// TIA Portal V17 export
// export: Created 2024-09-02T12:50:04.2483482Z, ExportSetting WithDefaults, DisplayName Totally Integrated Automation Portal, DisplayVersion V17, DisplayName TIA Portal Openness, DisplayVersion V17, DisplayName TIA Portal Version Control Interface, DisplayVersion V17, DisplayName STEP 7 Professional, DisplayVersion V17, DisplayName STEP 7 Safety, DisplayVersion V17, DisplayName WinCC Professional, DisplayVersion V17
FUNCTION "SysFC_RF300_Comunication" : Void   // FC801, LAD
TITLE = RF300 Commands / RF300 Befehle
{ S7_Optimized_Access := 'TRUE' }
AUTHOR : STEAM
FAMILY : MOBY
NAME : MOBY
VERSION : 0.1
// stored: AutoNumber true, IsIECCheckEnabled false, SetENOAutomatically false, UDAEnableTagReadback false
   VAR_INPUT
      SequenceNr : Int;   // Sequenznummer des Funktionsaufrufes (muss Eindeutig pro SLG sein) / Sequence number of function call (must be unique for each SLG)
      FunctionNr : Int;   // Funktionsanwahl 1 - lesen, 2- schreiben usw. / Function selection 1 - read, 2- write etc.
      Start : Bool;   // Funktionsanwahl "Lesen" / function selection "Read"
      Reset : Bool;
      ADR_MDS : Int;   // Adresse Datenträger (MDS) / Data carrier address (MDS)
      ByteLength : Int;   // Anzahl der Bytes / Number of bytes
   END_VAR
   VAR_OUTPUT
      FunktionOk : Bool;
   END_VAR
   VAR_IN_OUT
      MDS_Data : Variant;
      Command : "TypeMobyBefehle";
      Finish : Bool;   // Auftrag Fertig "Lesen / Order Finished "Read"
   END_VAR
   VAR_TEMP
      t_VKE0 : Bool;
      t_VKE1 : Bool;
      t_RetVal : Word;
      t_OrderLineReady : Bool;
      t_MainOrderReady : Bool;
      t_FaultBuffer : Bool;
      t_HugeBuffer : UDInt;
      t_TempDInt : DInt;
      t_Command_INIT : "TypeMobySequenz";
   END_VAR
   VAR_TEMP   // added for the SCL form of the ladder/FBD networks
      _w1 : Bool;
      _w2 : Bool;
      _w3 : Bool;
   END_VAR
BEGIN

REGION Network 1: INIT
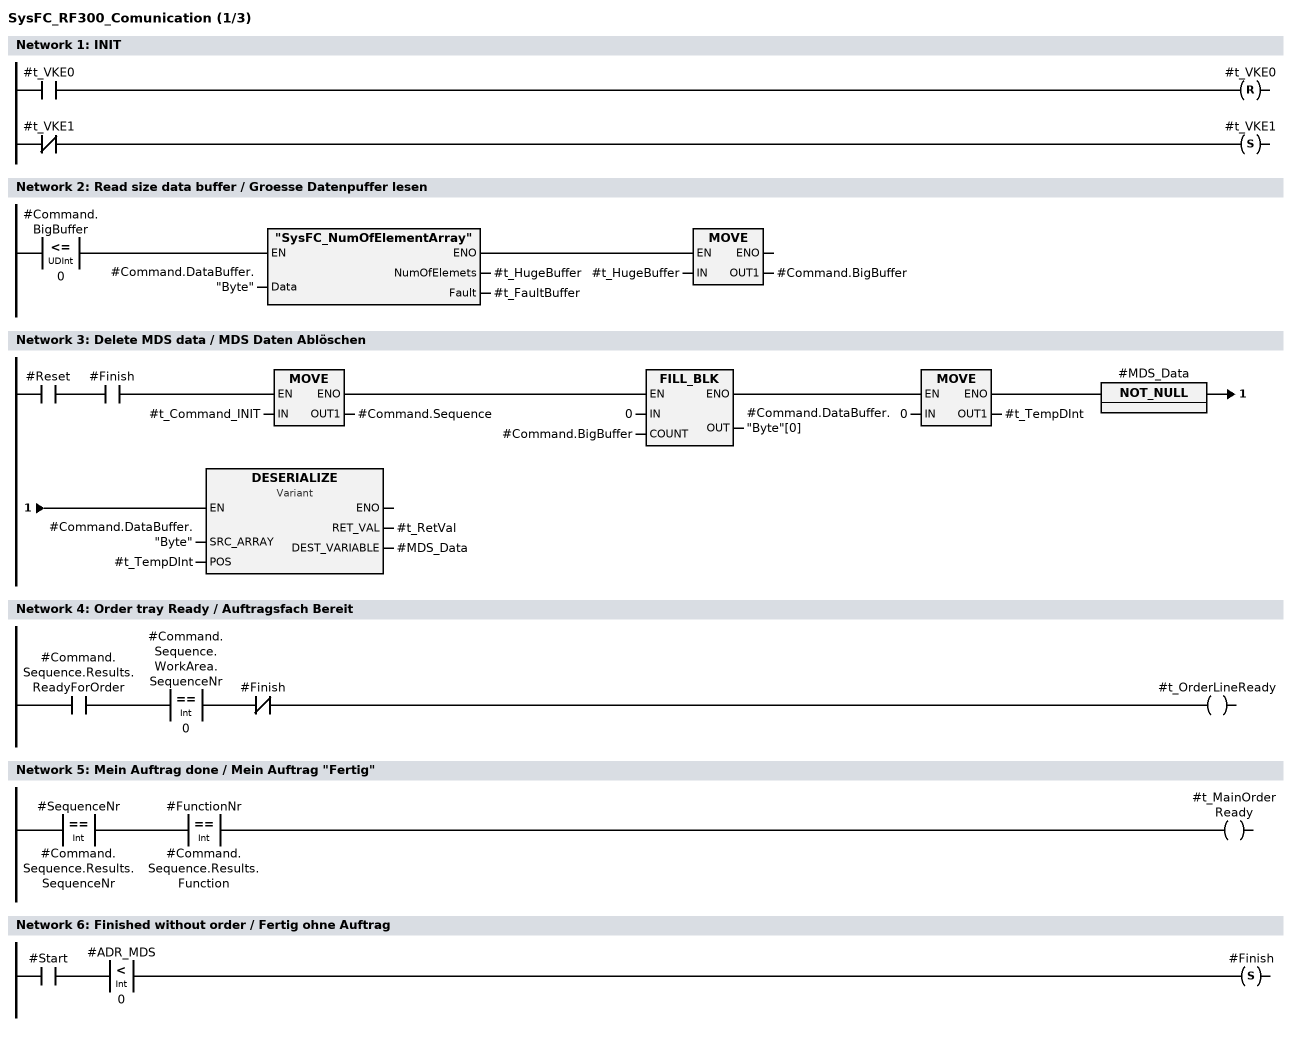
   RUNG wire#powerrail
      Contact( #t_VKE0 )
      R_Coil( #t_VKE0 )
   END_RUNG
   RUNG wire#powerrail
      I_Contact( #t_VKE1 )
      S_Coil( #t_VKE1 )
   END_RUNG
   // the same network as SCL:
   IF #t_VKE0 THEN #t_VKE0 := FALSE; END_IF;
   IF NOT #t_VKE1 THEN #t_VKE1 := TRUE; END_IF;
END_REGION

REGION Network 2: Read size data buffer / Groesse Datenpuffer lesen
   RUNG wire#powerrail
      { S7_Templates := "SrcType := UDInt" } LE_Contact(in1 := #Command.BigBuffer, in2 := 0)
      "SysFC_NumOfElementArray"(Data := #Command.DataBuffer."Byte", NumOfElemets => #t_HugeBuffer, Fault => #t_FaultBuffer)
      Move(in := #t_HugeBuffer, out1 => #Command.BigBuffer)
   END_RUNG
   // the same network as SCL:
   "SysFC_NumOfElementArray"(EN := #Command.BigBuffer <= 0,
                           Data := #Command.DataBuffer."Byte",
                           NumOfElemets => #t_HugeBuffer,
                           Fault => #t_FaultBuffer,
                           ENO => #_w1);
   IF #_w1 THEN #Command.BigBuffer := #t_HugeBuffer; END_IF;
END_REGION

REGION Network 3: Delete MDS data / MDS Daten Ablöschen
   // no SCL statement known for NOT_NULL: written as a call
   #_w1 := #Reset AND #Finish;
   IF #_w1 THEN
       #Command.Sequence := #t_Command_INIT;
       FILL_BLK(IN := 0, COUNT := #Command.BigBuffer, OUT => #Command.DataBuffer."Byte"[0]);
       #t_TempDInt := 0;
   END_IF;
   IF #_w1 AND NOT_NULL(#MDS_Data) THEN
       #t_RetVal := Deserialize(SRC_ARRAY := #Command.DataBuffer."Byte",
                               POS := #t_TempDInt,
                               DEST_VARIABLE => #MDS_Data);
   END_IF;
END_REGION

REGION Network 4: Order tray Ready / Auftragsfach Bereit
   RUNG wire#powerrail
      Contact( #Command.Sequence.Results.ReadyForOrder )
      { S7_Templates := "SrcType := Int" } EQ_Contact(in1 := #Command.Sequence.WorkArea.SequenceNr, in2 := 0)
      I_Contact( #Finish )
      Coil( #t_OrderLineReady )
   END_RUNG
   // the same network as SCL:
   #t_OrderLineReady := #Command.Sequence.Results.ReadyForOrder AND (#Command.Sequence.WorkArea.SequenceNr = 0) AND NOT #Finish;
END_REGION

REGION Network 5: Mein Auftrag done / Mein Auftrag "Fertig"
   RUNG wire#powerrail
      { S7_Templates := "SrcType := Int" } EQ_Contact(in1 := #SequenceNr, in2 := #Command.Sequence.Results.SequenceNr)
      { S7_Templates := "SrcType := Int" } EQ_Contact(in1 := #FunctionNr, in2 := #Command.Sequence.Results.Function)
      Coil( #t_MainOrderReady )
   END_RUNG
   // the same network as SCL:
   #t_MainOrderReady := (#SequenceNr = #Command.Sequence.Results.SequenceNr) AND (#FunctionNr = #Command.Sequence.Results.Function);
END_REGION

REGION Network 6: Finished without order / Fertig ohne Auftrag
   RUNG wire#powerrail
      Contact( #Start )
      { S7_Templates := "SrcType := Int" } LT_Contact(in1 := #ADR_MDS, in2 := 0)
      S_Coil( #Finish )
   END_RUNG
   // the same network as SCL:
   IF #Start AND (#ADR_MDS < 0) THEN #Finish := TRUE; END_IF;
END_REGION

REGION Network 7: Start job 'Read"; / Start Auftrag "Lesen"
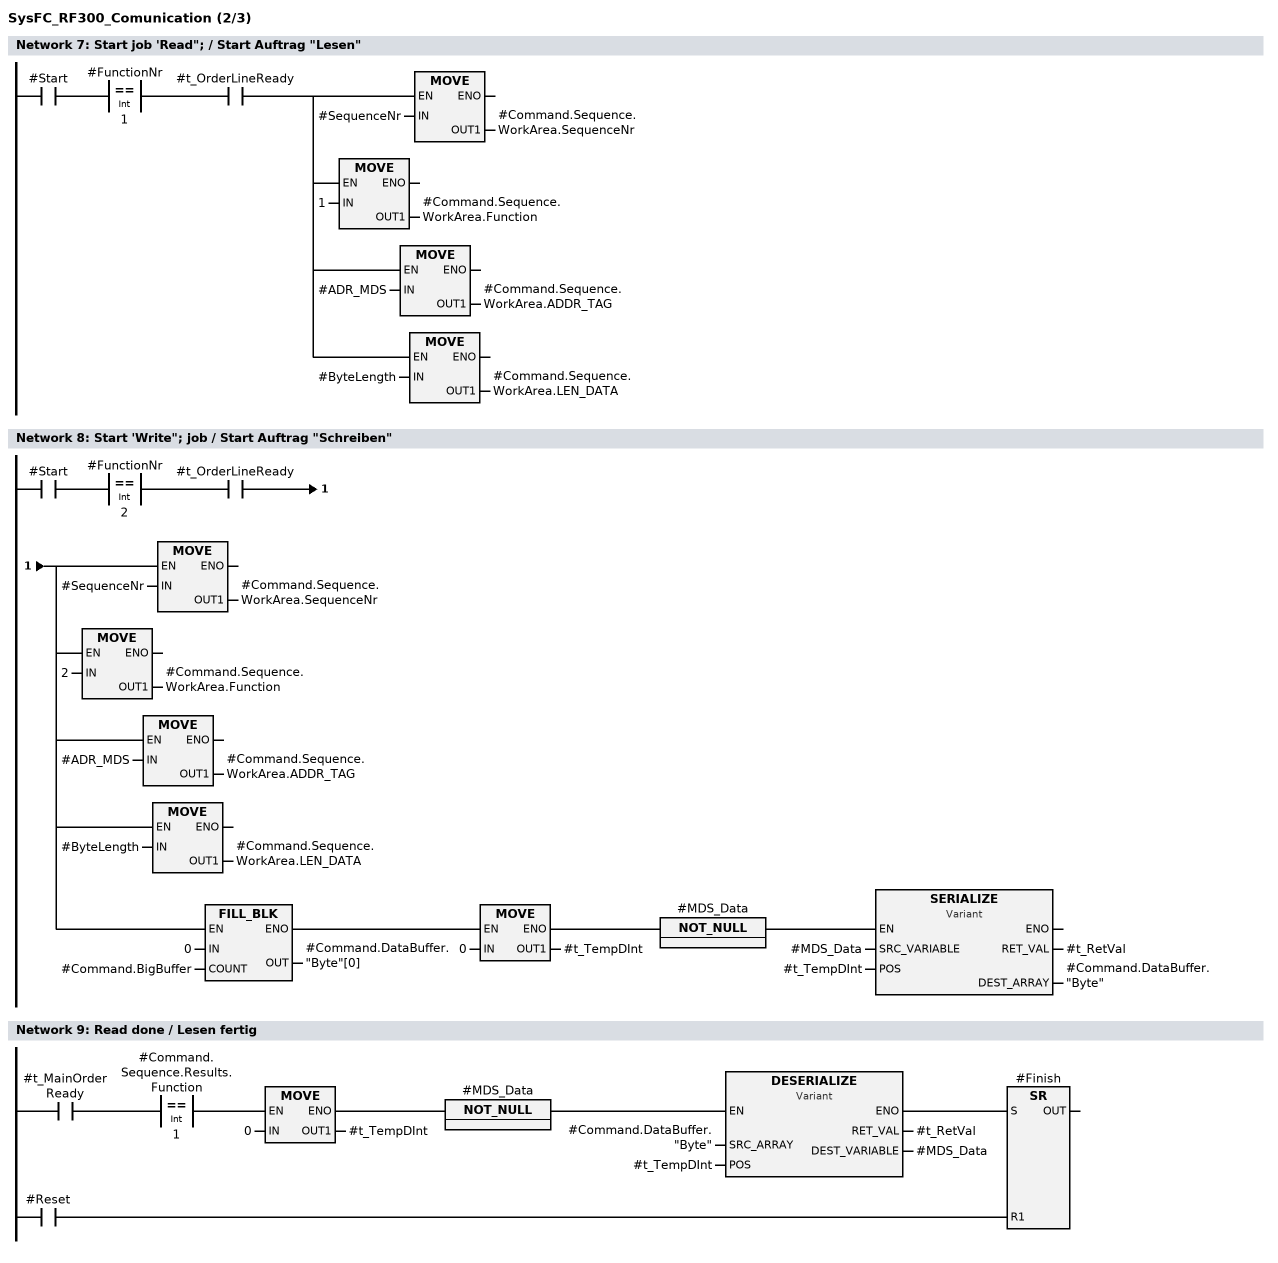
   RUNG wire#powerrail
      Contact( #Start )
      { S7_Templates := "SrcType := Int" } EQ_Contact(in1 := #FunctionNr, in2 := 1)
      Contact( #t_OrderLineReady )
      wire#w1
      Move(in := #SequenceNr, out1 => #Command.Sequence.WorkArea.SequenceNr)
   END_RUNG
   RUNG wire#w1
      Move(in := 1, out1 => #Command.Sequence.WorkArea.Function)
   END_RUNG
   RUNG wire#w1
      Move(in := #ADR_MDS, out1 => #Command.Sequence.WorkArea.ADDR_TAG)
   END_RUNG
   RUNG wire#w1
      Move(in := #ByteLength, out1 => #Command.Sequence.WorkArea.LEN_DATA)
   END_RUNG
   // the same network as SCL:
   IF #Start AND (#FunctionNr = 1) AND #t_OrderLineReady THEN
       #Command.Sequence.WorkArea.SequenceNr := #SequenceNr;
       #Command.Sequence.WorkArea.Function := 1;
       #Command.Sequence.WorkArea.ADDR_TAG := #ADR_MDS;
       #Command.Sequence.WorkArea.LEN_DATA := #ByteLength;
   END_IF;
END_REGION

REGION Network 8: Start 'Write"; job / Start Auftrag "Schreiben"
   // no SCL statement known for NOT_NULL: written as a call
   #_w1 := #Start AND (#FunctionNr = 2) AND #t_OrderLineReady;
   IF #_w1 THEN
       #Command.Sequence.WorkArea.SequenceNr := #SequenceNr;
       #Command.Sequence.WorkArea.Function := 2;
       #Command.Sequence.WorkArea.ADDR_TAG := #ADR_MDS;
       #Command.Sequence.WorkArea.LEN_DATA := #ByteLength;
       FILL_BLK(IN := 0, COUNT := #Command.BigBuffer, OUT => #Command.DataBuffer."Byte"[0]);
       #t_TempDInt := 0;
   END_IF;
   IF #_w1 AND NOT_NULL(#MDS_Data) THEN
       #t_RetVal := Serialize(SRC_VARIABLE := #MDS_Data,
                              POS := #t_TempDInt,
                              DEST_ARRAY => #Command.DataBuffer."Byte");
   END_IF;
END_REGION

REGION Network 9: Read done / Lesen fertig
   // no SCL statement known for NOT_NULL: written as a call
   #_w1 := #t_MainOrderReady AND (#Command.Sequence.Results.Function = 1);
   IF #_w1 THEN #t_TempDInt := 0; END_IF;
   #_w2 := #_w1 AND NOT_NULL(#MDS_Data);
   #t_RetVal := Deserialize(EN := #_w2,
                           SRC_ARRAY := #Command.DataBuffer."Byte",
                           POS := #t_TempDInt,
                           DEST_VARIABLE => #MDS_Data,
                           ENO => #_w3);
   IF #_w3 THEN
       #Finish := TRUE;   // SR flip-flop
   END_IF;
   IF #Reset THEN #Finish := FALSE; END_IF;
END_REGION

REGION Network 10: Write finished / Schreiben fertig
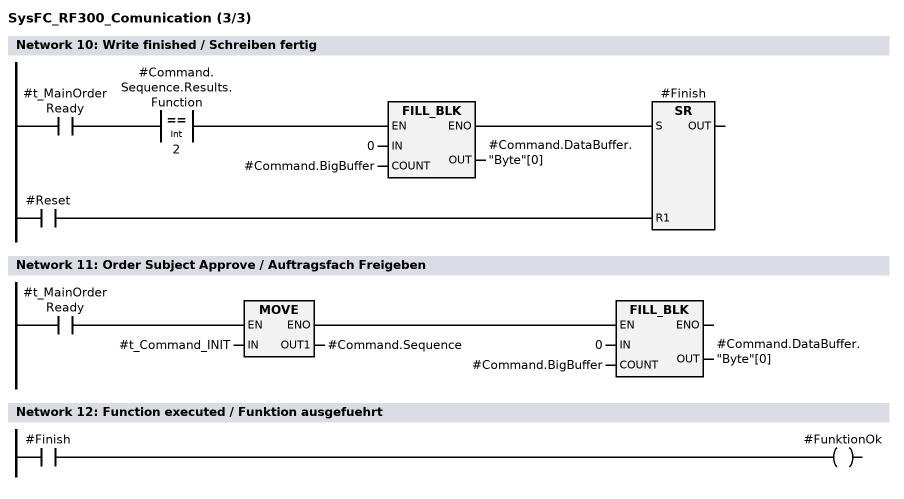
   RUNG wire#powerrail
      Contact( #t_MainOrderReady )
      { S7_Templates := "SrcType := Int" } EQ_Contact(in1 := #Command.Sequence.Results.Function, in2 := 2)
      FillBlockI(in := 0, count := #Command.BigBuffer, out => #Command.DataBuffer."Byte"[0])
      S_SR(operand := #Finish, r1 := wire#w1)
   END_RUNG
   RUNG wire#powerrail
      Contact( #Reset )
   END_RUNG wire#w1
   // the same network as SCL:
   #_w1 := #t_MainOrderReady AND (#Command.Sequence.Results.Function = 2);
   IF #_w1 THEN
       FILL_BLK(IN := 0, COUNT := #Command.BigBuffer, OUT => #Command.DataBuffer."Byte"[0]);
       #Finish := TRUE;   // SR flip-flop
   END_IF;
   IF #Reset THEN #Finish := FALSE; END_IF;
END_REGION

REGION Network 11: Order Subject Approve / Auftragsfach Freigeben
   RUNG wire#powerrail
      Contact( #t_MainOrderReady )
      Move(in := #t_Command_INIT, out1 => #Command.Sequence)
      FillBlockI(in := 0, count := #Command.BigBuffer, out => #Command.DataBuffer."Byte"[0])
   END_RUNG
   // the same network as SCL:
   IF #t_MainOrderReady THEN
       #Command.Sequence := #t_Command_INIT;
       FILL_BLK(IN := 0, COUNT := #Command.BigBuffer, OUT => #Command.DataBuffer."Byte"[0]);
   END_IF;
END_REGION

REGION Network 12: Function executed / Funktion ausgefuehrt
   RUNG wire#powerrail
      Contact( #Finish )
      Coil( #FunktionOk )
   END_RUNG
   // the same network as SCL:
   #FunktionOk := #Finish;
END_REGION
END_FUNCTION
